(* IEC 61131-3 sources: TIA2AX/tests/V18/test_projects/expected/HW_2000528_main/PLC_LINE_L, 7 files *)

(* ---- HwIdentifiers.st ---- *)
TYPE
	HwIdentifiers : WORD
	(
		PLC_LINE_L_Rail_0 :=	WORD#256,
		PLC_LINE_L :=	WORD#48,
		PLC_LINE_L_Card_reader_writer_1 :=	WORD#51,
		PLC_LINE_L_CPU_display_1 :=	WORD#54,
		PLC_LINE_L_OPC_UA_1 :=	WORD#117,
		PLC_LINE_L_DP_interface_1 :=	WORD#60,
		PLC_LINE_L_PROFINET_interface_1 :=	WORD#64,
		PLC_LINE_L_PROFINET_interface_1_Port_1 :=	WORD#65,
		PLC_LINE_L_PROFINET_interface_1_Port_2 :=	WORD#66,
		PLC_LINE_L_PROFINET_interface_2 :=	WORD#72,
		PLC_LINE_L_PROFINET_interface_2_Port_1 :=	WORD#73,
		UR5_st4_L_Rack :=	WORD#273,
		UR5_st4_L :=	WORD#258,
		UR5_st4_L_Interface :=	WORD#259,
		UR5_st4_L_Interface_RJ45_10_100_MBit_s :=	WORD#260,
		UR5_st4_L_V1_0 :=	WORD#261,
		UR5_st4_L_1_T2O_State :=	WORD#262,
		UR5_st4_L_2_T2O_IO :=	WORD#263,
		UR5_st4_L_3_T2O_Joints :=	WORD#264,
		UR5_st4_L_4_T2O_TCP :=	WORD#265,
		UR5_st4_L_5_T2O_General_Purpose_Bit_Registers :=	WORD#266,
		UR5_st4_L_6_T2O_General_Purpose_Int_Registers :=	WORD#267,
		UR5_st4_L_7_T2O_General_Purpose_Float_Registers :=	WORD#268,
		UR5_st4_L_8_O2T_Robot_IO :=	WORD#269,
		UR5_st4_L_9_O2T_General_Purpose_Registers_1 :=	WORD#270,
		UR5_st4_L_10_O2T_General_Purpose_Registers_2 :=	WORD#271,
		WP001_DM260_L_Rack :=	WORD#275,
		WP001_DM260_L :=	WORD#276,
		WP001_DM260_L_Interface :=	WORD#277,
		WP001_DM260_L_Interface_Port_1 :=	WORD#278,
		WP001_DM260_L_DataMan_260 :=	WORD#279,
		WP001_DM260_L_Acquisition_Control_1 :=	WORD#280,
		WP001_DM260_L_Acquisition_Status_1 :=	WORD#281,
		WP001_DM260_L_Results_Control_1 :=	WORD#282,
		WP001_DM260_L_Results_Status_1 :=	WORD#283,
		WP001_DM260_L_Soft_Event_Control_1 :=	WORD#284,
		WP001_DM260_L_User_Data_64_bytes_1 :=	WORD#285,
		WP001_DM260_L_Result_Data_64_bytes_1 :=	WORD#286,
		R5A1_L_Rack_0 :=	WORD#288,
		R5A1_L :=	WORD#289,
		R5A1_L_R5A1_L :=	WORD#290,
		R5A1_L_PROFINET_interface :=	WORD#291,
		R5A1_L_PROFINET_interface_Port_1 :=	WORD#293,
		R5A1_L_PROFINET_interface_Port_2 :=	WORD#292,
		R5A1_L_BA_2xRJ45 :=	WORD#293,
		R5A1_L_CM_PtP_1 :=	WORD#294,
		R5A1_L_AI_4xU_I_2_wire_ST_1 :=	WORD#295,
		R5A1_L_AI_4xU_I_2_wire_ST_2 :=	WORD#296,
		R5A1_L_AQ_4xU_I_ST_1 :=	WORD#297,
		R5A1_L_DI_16x24VDC_ST_1 :=	WORD#298,
		R5A1_L_DI_16x24VDC_ST_2 :=	WORD#299,
		R5A1_L_DI_16x24VDC_ST_3 :=	WORD#300,
		R5A1_L_DI_16x24VDC_ST_4 :=	WORD#301,
		R5A1_L_DI_16x24VDC_ST_5 :=	WORD#302,
		R5A1_L_DQ_16x24VDC_0_5A_ST_1 :=	WORD#303,
		R5A1_L_DQ_16x24VDC_0_5A_ST_2 :=	WORD#304,
		R5A1_L_DQ_16x24VDC_0_5A_ST_3 :=	WORD#305,
		R5A1_L_DQ_16x24VDC_0_5A_ST_4 :=	WORD#306,
		R5A1_L_TM_Pulse_2x24V_1 :=	WORD#307,
		R5A1_L_TM_Pulse_2x24V_2 :=	WORD#308,
		R5A1_L_Server_module_1 :=	WORD#309,
		R0_L_Rack_0 :=	WORD#311,
		R0_L :=	WORD#312,
		R0_L_R0_L :=	WORD#313,
		R0_L_PROFINET_interface :=	WORD#314,
		R0_L_PROFINET_interface_Port_1 :=	WORD#316,
		R0_L_PROFINET_interface_Port_2 :=	WORD#315,
		R0_L_BA_2xRJ45 :=	WORD#316,
		R0_L_DI_16x24VDC_ST_1 :=	WORD#317,
		R0_L_DI_16x24VDC_ST_2 :=	WORD#318,
		R0_L_DI_16x24VDC_ST_3 :=	WORD#319,
		R0_L_DI_16x24VDC_ST_4 :=	WORD#320,
		R0_L_DI_16x24VDC_ST_5 :=	WORD#321,
		R0_L_DI_16x24VDC_ST_6 :=	WORD#322,
		R0_L_DQ_16x24VDC_0_5A_ST_1 :=	WORD#323,
		R0_L_DQ_16x24VDC_0_5A_ST_2 :=	WORD#324,
		R0_L_DQ_16x24VDC_0_5A_ST_3 :=	WORD#325,
		R0_L_DQ_16x24VDC_0_5A_ST_4 :=	WORD#326,
		R0_L_DQ_16x24VDC_0_5A_ST_5 :=	WORD#327,
		R0_L_DI_8x24VDC_ST_1 :=	WORD#328,
		R0_L_DI_8x24VDC_ST_2 :=	WORD#329,
		R0_L_DI_8x24VDC_ST_3 :=	WORD#330,
		R0_L_DI_8x24VDC_ST_4 :=	WORD#331,
		R0_L_DI_16x24VDC_ST_7 :=	WORD#332,
		R0_L_Server_module_1 :=	WORD#333,
		R1A1_L_Rack_0 :=	WORD#335,
		R1A1_L :=	WORD#336,
		R1A1_L_R1A1_L :=	WORD#337,
		R1A1_L_PROFINET_interface :=	WORD#338,
		R1A1_L_PROFINET_interface_Port_1 :=	WORD#340,
		R1A1_L_PROFINET_interface_Port_2 :=	WORD#339,
		R1A1_L_BA_2xRJ45 :=	WORD#340,
		R1A1_L_DI_16x24VDC_ST_1 :=	WORD#341,
		R1A1_L_DI_16x24VDC_ST_2 :=	WORD#342,
		R1A1_L_DI_16x24VDC_ST_3 :=	WORD#343,
		R1A1_L_DI_16x24VDC_ST_4 :=	WORD#344,
		R1A1_L_DQ_16x24VDC_0_5A_ST_1 :=	WORD#345,
		R1A1_L_DQ_16x24VDC_0_5A_ST_2 :=	WORD#346,
		R1A1_L_DQ_16x24VDC_0_5A_ST_3 :=	WORD#347,
		R1A1_L_Server_module_1 :=	WORD#348,
		R2A1_L_Rack_0 :=	WORD#350,
		R2A1_L :=	WORD#351,
		R2A1_L_R2A1_L :=	WORD#352,
		R2A1_L_PROFINET_interface :=	WORD#353,
		R2A1_L_PROFINET_interface_Port_1 :=	WORD#355,
		R2A1_L_PROFINET_interface_Port_2 :=	WORD#354,
		R2A1_L_BA_2xRJ45 :=	WORD#355,
		R2A1_L_AI_4xU_I_2_wire_ST_1 :=	WORD#356,
		R2A1_L_DI_16x24VDC_ST_1 :=	WORD#357,
		R2A1_L_DI_16x24VDC_ST_2 :=	WORD#358,
		R2A1_L_DI_16x24VDC_ST_3 :=	WORD#359,
		R2A1_L_DI_16x24VDC_ST_4 :=	WORD#360,
		R2A1_L_DI_16x24VDC_ST_5 :=	WORD#361,
		R2A1_L_DI_16x24VDC_ST_6 :=	WORD#362,
		R2A1_L_DQ_16x24VDC_0_5A_ST_1 :=	WORD#363,
		R2A1_L_DQ_16x24VDC_0_5A_ST_2 :=	WORD#364,
		R2A1_L_DQ_16x24VDC_0_5A_ST_3 :=	WORD#365,
		R2A1_L_TM_Pulse_2x24V_1 :=	WORD#366,
		R2A1_L_Server_module_1 :=	WORD#367,
		R6_L_Rack_0 :=	WORD#369,
		R6_L :=	WORD#370,
		R6_L_R6_L :=	WORD#371,
		R6_L_PROFINET_interface :=	WORD#372,
		R6_L_PROFINET_interface_Port_1 :=	WORD#374,
		R6_L_PROFINET_interface_Port_2 :=	WORD#373,
		R6_L_BA_2xRJ45 :=	WORD#374,
		R6_L_DI_16x24VDC_ST_1 :=	WORD#375,
		R6_L_DI_16x24VDC_ST_2 :=	WORD#376,
		R6_L_DQ_16x24VDC_0_5A_ST_1 :=	WORD#377,
		R6_L_DQ_16x24VDC_0_5A_ST_2 :=	WORD#378,
		R6_L_Server_module_1 :=	WORD#379,
		WP002_DM260_L_Rack :=	WORD#381,
		WP002_DM260_L :=	WORD#382,
		WP002_DM260_L_Interface :=	WORD#383,
		WP002_DM260_L_Interface_Port_1 :=	WORD#384,
		WP002_DM260_L_DataMan_260 :=	WORD#385,
		WP002_DM260_L_Acquisition_Control_1 :=	WORD#386,
		WP002_DM260_L_Acquisition_Status_1 :=	WORD#387,
		WP002_DM260_L_Results_Control_1 :=	WORD#388,
		WP002_DM260_L_Results_Status_1 :=	WORD#389,
		WP002_DM260_L_Soft_Event_Control_1 :=	WORD#390,
		WP002_DM260_L_User_Data_64_bytes_1 :=	WORD#391,
		WP002_DM260_L_Result_Data_64_bytes_1 :=	WORD#392,
		CPX_WP5_L_PN_IO_Interface :=	WORD#396,
		CPX_WP5_L_PN_IO_Interface_Port_1 :=	WORD#397,
		CPX_WP5_L_PN_IO_Interface_Port_2 :=	WORD#398,
		CPX_WP5_L_CPX_Rev_30 :=	WORD#399,
		CPX_WP5_L_FB33_PNIO_Module_1 :=	WORD#400,
		CPX_WP5_L_MPA1S_VMPA1_FB_EMS_8_8DO_1 :=	WORD#401,
		CPX_WP5_L_MPA1S_VMPA1_FB_EMS_8_8DO_2 :=	WORD#402,
		CPX_WP5_L_MPA1S_VMPA1_FB_EMS_8_8DO_3 :=	WORD#403,
		CPX_TS_L_PN_IO_Interface :=	WORD#407,
		CPX_TS_L_PN_IO_Interface_Port_1 :=	WORD#408,
		CPX_TS_L_PN_IO_Interface_Port_2 :=	WORD#409,
		CPX_TS_L_CPX_Rev_30 :=	WORD#410,
		CPX_TS_L_FB33_PNIO_Module_1 :=	WORD#411,
		CPX_TS_L_MPA2S_VMPA2_FB_EMS_4_4DO_1 :=	WORD#412,
		CPX_TS_L_MPA2G_VMPA2_FB_EMG_4_4DO_1 :=	WORD#413,
		CPX_TS_L_MPA1G_VMPA1_FB_EMG_8_8DO_2 :=	WORD#414,
		CPX_TS_L_MPA1G_VMPA1_FB_EMG_8_8DO_3 :=	WORD#415,
		CPX_TS_L_MPA1G_VMPA1_FB_EMG_8_8DO_4 :=	WORD#416,
		CPX_TS_L_MPA1G_VMPA1_FB_EMG_8_8DO_5 :=	WORD#417,
		CPX_TS_L_MPA1G_VMPA1_FB_EMG_8_8DO_6 :=	WORD#418,
		CPX_WP2_L_PN_IO_Interface :=	WORD#422,
		CPX_WP2_L_PN_IO_Interface_Port_1 :=	WORD#423,
		CPX_WP2_L_PN_IO_Interface_Port_2 :=	WORD#424,
		CPX_WP2_L_CPX_Rev_30 :=	WORD#425,
		CPX_WP2_L_FB33_PNIO_Module_1 :=	WORD#426,
		CPX_WP2_L_MPA1S_VMPA1_FB_EMS_8_8DO_1 :=	WORD#427,
		CPX_WP2_L_MPA1S_VMPA1_FB_EMS_8_8DO_2 :=	WORD#428,
		CPX_WP2_L_MPA1S_VMPA1_FB_EMS_8_8DO_3 :=	WORD#429,
		CPX_WP2_L_MPA1G_VMPA1_FB_EMG_8_8DO_3 :=	WORD#430,
		fx0_gpnt_L_FX0_GPNT_V2 :=	WORD#434,
		fx0_gpnt_L_FX0_GPNT_V2_Port_1 :=	WORD#435,
		fx0_gpnt_L_FX0_GPNT_V2_Port_2 :=	WORD#436,
		fx0_gpnt_L_FX0_GPNT_V2_1 :=	WORD#437,
		fx0_gpnt_L_Input_Data_Block_1_1 :=	WORD#438,
		fx0_gpnt_L_Input_Data_Block_2_1 :=	WORD#439,
		fx0_gpnt_L_Input_Data_Block_3_1 :=	WORD#440,
		fx0_gpnt_L_Input_Data_Block_4_1 :=	WORD#441,
		fx0_gpnt_L_Input_Data_Block_5_1 :=	WORD#442,
		fx0_gpnt_L_Output_Data_Block_1_1 :=	WORD#443,
		fx0_gpnt_L_Output_Data_Block_2_1 :=	WORD#444,
		fx0_gpnt_L_Output_Data_Block_3_1 :=	WORD#445,
		fx0_gpnt_L_Output_Data_Block_4_1 :=	WORD#446,
		fx0_gpnt_L_Output_Data_Block_5_1 :=	WORD#447,
		WP004_DM260_L_Rack :=	WORD#449,
		WP004_DM260_L :=	WORD#450,
		WP004_DM260_L_Interface :=	WORD#451,
		WP004_DM260_L_Interface_Port_1 :=	WORD#452,
		WP004_DM260_L_DataMan_260 :=	WORD#453,
		WP004_DM260_L_Acquisition_Control_1 :=	WORD#454,
		WP004_DM260_L_Acquisition_Status_1 :=	WORD#455,
		WP004_DM260_L_Results_Control_1 :=	WORD#456,
		WP004_DM260_L_Results_Status_1 :=	WORD#457,
		WP004_DM260_L_Soft_Event_Control_1 :=	WORD#458,
		WP004_DM260_L_User_Data_64_bytes_1 :=	WORD#459,
		WP004_DM260_L_Result_Data_64_bytes_1 :=	WORD#460,
		WP0031_DM260_L_Rack :=	WORD#462,
		WP0031_DM260_L :=	WORD#463,
		WP0031_DM260_L_Interface :=	WORD#464,
		WP0031_DM260_L_Interface_Port_1 :=	WORD#465,
		WP0031_DM260_L_DataMan_260 :=	WORD#466,
		WP0031_DM260_L_Acquisition_Control_1 :=	WORD#467,
		WP0031_DM260_L_Acquisition_Status_1 :=	WORD#468,
		WP0031_DM260_L_Results_Control_1 :=	WORD#469,
		WP0031_DM260_L_Results_Status_1 :=	WORD#470,
		WP0031_DM260_L_Soft_Event_Control_1 :=	WORD#471,
		WP0031_DM260_L_User_Data_64_bytes_1 :=	WORD#472,
		WP0031_DM260_L_Result_Data_64_bytes_1 :=	WORD#473,
		WP003_DM260_L_Rack :=	WORD#475,
		WP003_DM260_L :=	WORD#476,
		WP003_DM260_L_Interface :=	WORD#477,
		WP003_DM260_L_Interface_Port_1 :=	WORD#478,
		WP003_DM260_L_DataMan_260 :=	WORD#479,
		WP003_DM260_L_Acquisition_Control_1 :=	WORD#480,
		WP003_DM260_L_Acquisition_Status_1 :=	WORD#481,
		WP003_DM260_L_Results_Control_1 :=	WORD#482,
		WP003_DM260_L_Results_Status_1 :=	WORD#483,
		WP003_DM260_L_Soft_Event_Control_1 :=	WORD#484,
		WP003_DM260_L_User_Data_64_bytes_1 :=	WORD#485,
		WP003_DM260_L_Result_Data_64_bytes_1 :=	WORD#486,
		WP005_DM260_L_Rack :=	WORD#488,
		WP005_DM260_L :=	WORD#489,
		WP005_DM260_L_Interface :=	WORD#490,
		WP005_DM260_L_Interface_Port_1 :=	WORD#491,
		WP005_DM260_L_DataMan_260 :=	WORD#492,
		WP005_DM260_L_Acquisition_Control_1 :=	WORD#493,
		WP005_DM260_L_Acquisition_Status_1 :=	WORD#494,
		WP005_DM260_L_Results_Control_1 :=	WORD#495,
		WP005_DM260_L_Results_Status_1 :=	WORD#496,
		WP005_DM260_L_Soft_Event_Control_1 :=	WORD#497,
		WP005_DM260_L_User_Data_64_bytes_1 :=	WORD#498,
		WP005_DM260_L_Result_Data_64_bytes_1 :=	WORD#499,
		WP006_DM260_L_Rack :=	WORD#501,
		WP006_DM260_L :=	WORD#502,
		WP006_DM260_L_Interface :=	WORD#503,
		WP006_DM260_L_Interface_Port_1 :=	WORD#504,
		WP006_DM260_L_DataMan_260 :=	WORD#505,
		WP006_DM260_L_Acquisition_Control_1 :=	WORD#506,
		WP006_DM260_L_Acquisition_Status_1 :=	WORD#507,
		WP006_DM260_L_Results_Control_1 :=	WORD#508,
		WP006_DM260_L_Results_Status_1 :=	WORD#509,
		WP006_DM260_L_Soft_Event_Control_1 :=	WORD#510,
		WP006_DM260_L_User_Data_64_bytes_1 :=	WORD#511,
		WP006_DM260_L_Result_Data_64_bytes_1 :=	WORD#512,
		WP001_DM8050_L_Rack :=	WORD#514,
		WP001_DM8050_L :=	WORD#515,
		WP001_DM8050_L_Interface :=	WORD#516,
		WP001_DM8050_L_Interface_Port_1 :=	WORD#517,
		WP001_DM8050_L_DataMan_8000 :=	WORD#518,
		WP001_DM8050_L_Acquisition_Control_1 :=	WORD#519,
		WP001_DM8050_L_Acquisition_Status_1 :=	WORD#520,
		WP001_DM8050_L_Results_Control_1 :=	WORD#521,
		WP001_DM8050_L_Results_Status_1 :=	WORD#522,
		WP001_DM8050_L_Soft_Event_Control_1 :=	WORD#523,
		WP001_DM8050_L_User_Data_64_bytes_1 :=	WORD#524,
		WP001_DM8050_L_Result_Data_64_bytes_1 :=	WORD#525,
		WP004_DM8050_L_Rack :=	WORD#527,
		WP004_DM8050_L :=	WORD#528,
		WP004_DM8050_L_Interface :=	WORD#529,
		WP004_DM8050_L_Interface_Port_1 :=	WORD#530,
		WP004_DM8050_L_DataMan_8000 :=	WORD#531,
		WP004_DM8050_L_Acquisition_Control_1 :=	WORD#532,
		WP004_DM8050_L_Acquisition_Status_1 :=	WORD#533,
		WP004_DM8050_L_Results_Control_1 :=	WORD#534,
		WP004_DM8050_L_Results_Status_1 :=	WORD#535,
		WP004_DM8050_L_Soft_Event_Control_1 :=	WORD#536,
		WP004_DM8050_L_User_Data_64_bytes_1 :=	WORD#537,
		WP004_DM8050_L_Result_Data_64_bytes_1 :=	WORD#538,
		WP003_CAM_L_Rack :=	WORD#540,
		WP003_CAM_L :=	WORD#541,
		WP003_CAM_L_Interface :=	WORD#542,
		WP003_CAM_L_Interface_Port_1 :=	WORD#543,
		WP003_CAM_L_In_Sight_IS2XXX_CC_B :=	WORD#544,
		WP003_CAM_L_Acquisition_Control_1 :=	WORD#545,
		WP003_CAM_L_Acquisition_Status_1 :=	WORD#546,
		WP003_CAM_L_Inspection_Control_1 :=	WORD#547,
		WP003_CAM_L_Inspection_Status_1 :=	WORD#548,
		WP003_CAM_L_Command_Control_1 :=	WORD#549,
		WP003_CAM_L_SoftEvent_Control_1 :=	WORD#550,
		WP003_CAM_L_User_Data_64_bytes_1 :=	WORD#551,
		WP003_CAM_L_Results_64_bytes_1 :=	WORD#552,
		WP004_CAM_L_Rack :=	WORD#554,
		WP004_CAM_L :=	WORD#555,
		WP004_CAM_L_Interface :=	WORD#556,
		WP004_CAM_L_Interface_Port_1 :=	WORD#557,
		WP004_CAM_L_In_Sight_IS2XXX_CC_B :=	WORD#558,
		WP004_CAM_L_Acquisition_Control_1 :=	WORD#559,
		WP004_CAM_L_Acquisition_Status_1 :=	WORD#560,
		WP004_CAM_L_Inspection_Control_1 :=	WORD#561,
		WP004_CAM_L_Inspection_Status_1 :=	WORD#562,
		WP004_CAM_L_Command_Control_1 :=	WORD#563,
		WP004_CAM_L_SoftEvent_Control_1 :=	WORD#564,
		WP004_CAM_L_User_Data_64_bytes_1 :=	WORD#565,
		WP004_CAM_L_Results_64_bytes_1 :=	WORD#566,
		WP0031_DM8700_L_Rack :=	WORD#568,
		WP0031_DM8700_L :=	WORD#569,
		WP0031_DM8700_L_Interface :=	WORD#570,
		WP0031_DM8700_L_Interface_Port_1 :=	WORD#571,
		WP0031_DM8700_L_DataMan_8700_CC_B :=	WORD#572,
		WP0031_DM8700_L_Acquisition_Control_1 :=	WORD#573,
		WP0031_DM8700_L_Acquisition_Status_1 :=	WORD#574,
		WP0031_DM8700_L_Results_Control_1 :=	WORD#575,
		WP0031_DM8700_L_Results_Status_1 :=	WORD#576,
		WP0031_DM8700_L_Soft_Event_Control_1 :=	WORD#577,
		WP0031_DM8700_L_User_Data_64_bytes_1 :=	WORD#578,
		WP0031_DM8700_L_Result_Data_64_bytes_1 :=	WORD#579,
		WP002_DM8050_L_Rack :=	WORD#581,
		WP002_DM8050_L :=	WORD#582,
		WP002_DM8050_L_Interface :=	WORD#583,
		WP002_DM8050_L_Interface_Port_1 :=	WORD#584,
		WP002_DM8050_L_DataMan_8000 :=	WORD#585,
		WP002_DM8050_L_Acquisition_Control_1 :=	WORD#586,
		WP002_DM8050_L_Acquisition_Status_1 :=	WORD#587,
		WP002_DM8050_L_Results_Control_1 :=	WORD#588,
		WP002_DM8050_L_Results_Status_1 :=	WORD#589,
		WP002_DM8050_L_Soft_Event_Control_1 :=	WORD#590,
		WP002_DM8050_L_User_Data_64_bytes_1 :=	WORD#591,
		WP002_DM8050_L_Result_Data_64_bytes_1 :=	WORD#592,
		CPX_Rack_L_PN_IO_Interface :=	WORD#596,
		CPX_Rack_L_PN_IO_Interface_Port_1 :=	WORD#597,
		CPX_Rack_L_PN_IO_Interface_Port_2 :=	WORD#598,
		CPX_Rack_L_CPX_Rev_30 :=	WORD#599,
		CPX_Rack_L_FB33_PNIO_Module_1 :=	WORD#600,
		CPX_Rack_L_16DI_16DI_1 :=	WORD#601,
		CPX_Rack_L_16DI_16DI_2 :=	WORD#602,
		CPX_Rack_L_16DI_16DI_3 :=	WORD#603,
		CPX_Rack_L_16DI_16DI_4 :=	WORD#604,
		CPX_Rack_L_16DI_16DI_5 :=	WORD#605,
		CPX_Rack_L_MPA1S_VMPA1_FB_EMS_8_8DO_1 :=	WORD#606,
		CPX_Rack_L_MPA1S_VMPA1_FB_EMS_8_8DO_2 :=	WORD#607,
		CPX_Rack_L_MPA1S_VMPA1_FB_EMS_8_8DO_3 :=	WORD#608,
		CPX_Rack_L_MPA1S_VMPA1_FB_EMS_8_8DO_4 :=	WORD#609,
		CPX_Rack_L_MPA1S_VMPA1_FB_EMS_8_8DO_5 :=	WORD#610,
		WP000_DM260_L_Rack :=	WORD#612,
		WP000_DM260_L :=	WORD#613,
		WP000_DM260_L_Interface :=	WORD#614,
		WP000_DM260_L_Interface_Port_1 :=	WORD#615,
		WP000_DM260_L_DataMan_260 :=	WORD#616,
		WP000_DM260_L_Acquisition_Control_1 :=	WORD#617,
		WP000_DM260_L_Acquisition_Status_1 :=	WORD#618,
		WP000_DM260_L_Results_Control_1 :=	WORD#619,
		WP000_DM260_L_Results_Status_1 :=	WORD#620,
		WP000_DM260_L_Soft_Event_Control_1 :=	WORD#621,
		WP000_DM260_L_User_Data_64_bytes_1 :=	WORD#622,
		WP000_DM260_L_Result_Data_64_bytes_1 :=	WORD#623,
		WP000_DM8050_L_Rack :=	WORD#625,
		WP000_DM8050_L :=	WORD#626,
		WP000_DM8050_L_Interface :=	WORD#627,
		WP000_DM8050_L_Interface_Port_1 :=	WORD#628,
		WP000_DM8050_L_DataMan_8000 :=	WORD#629,
		WP000_DM8050_L_Acquisition_Control_1 :=	WORD#630,
		WP000_DM8050_L_Acquisition_Status_1 :=	WORD#631,
		WP000_DM8050_L_Results_Control_1 :=	WORD#632,
		WP000_DM8050_L_Results_Status_1 :=	WORD#633,
		WP000_DM8050_L_Soft_Event_Control_1 :=	WORD#634,
		WP000_DM8050_L_User_Data_64_bytes_1 :=	WORD#635,
		WP000_DM8050_L_Result_Data_64_bytes_1 :=	WORD#636,
		NONE:= WORD#0
	);
END_TYPE

(* ---- HwInputs.st ---- *)
TYPE
	HwInputs : STRUCT
		UR5_st4_L_1_T2O_State AT %B1080 : ARRAY[0..31] OF BYTE;
		UR5_st4_L_2_T2O_IO AT %B1112 : ARRAY[0..67] OF BYTE;
		UR5_st4_L_3_T2O_Joints AT %B2696 : ARRAY[0..103] OF BYTE;
		UR5_st4_L_4_T2O_TCP AT %B1304 : ARRAY[0..75] OF BYTE;
		UR5_st4_L_5_T2O_General_Purpose_Bit_Registers AT %B1380 : ARRAY[0..7] OF BYTE;
		UR5_st4_L_6_T2O_General_Purpose_Int_Registers AT %B2800 : ARRAY[0..95] OF BYTE;
		UR5_st4_L_7_T2O_General_Purpose_Float_Registers AT %B2896 : ARRAY[0..95] OF BYTE;
		WP001_DM260_L_Acquisition_Status_1 AT %B5100 : ARRAY[0..2] OF BYTE;
		WP001_DM260_L_Results_Status_1 AT %B5103 : BYTE;
		WP001_DM260_L_Soft_Event_Control_1 AT %B5104 : BYTE;
		WP001_DM260_L_Result_Data_64_bytes_1 AT %B5110 : ARRAY[0..71] OF BYTE;
		R5A1_L_CM_PtP_1 AT %B270 : ARRAY[0..7] OF BYTE;
		R5A1_L_AI_4xU_I_2_wire_ST_1 AT %B278 : ARRAY[0..7] OF BYTE;
		R5A1_L_AI_4xU_I_2_wire_ST_2 AT %B286 : ARRAY[0..7] OF BYTE;
		R5A1_L_DI_16x24VDC_ST_1 AT %B20 : WORD;
		R5A1_L_DI_16x24VDC_ST_2 AT %B22 : WORD;
		R5A1_L_DI_16x24VDC_ST_3 AT %B24 : WORD;
		R5A1_L_DI_16x24VDC_ST_4 AT %B26 : WORD;
		R5A1_L_DI_16x24VDC_ST_5 AT %B28 : WORD;
		R5A1_L_TM_Pulse_2x24V_1 AT %B224 : ARRAY[0..15] OF BYTE;
		R5A1_L_TM_Pulse_2x24V_2 AT %B250 : ARRAY[0..15] OF BYTE;
		R0_L_DI_16x24VDC_ST_1 AT %B0 : WORD;
		R0_L_DI_16x24VDC_ST_2 AT %B2 : WORD;
		R0_L_DI_16x24VDC_ST_3 AT %B4 : WORD;
		R0_L_DI_16x24VDC_ST_4 AT %B6 : WORD;
		R0_L_DI_16x24VDC_ST_5 AT %B8 : WORD;
		R0_L_DI_16x24VDC_ST_6 AT %B10 : WORD;
		R0_L_DI_8x24VDC_ST_1 AT %B12 : BYTE;
		R0_L_DI_8x24VDC_ST_2 AT %B13 : BYTE;
		R0_L_DI_8x24VDC_ST_3 AT %B14 : BYTE;
		R0_L_DI_8x24VDC_ST_4 AT %B15 : BYTE;
		R0_L_DI_16x24VDC_ST_7 AT %B16 : WORD;
		R1A1_L_DI_16x24VDC_ST_1 AT %B100 : WORD;
		R1A1_L_DI_16x24VDC_ST_2 AT %B102 : WORD;
		R1A1_L_DI_16x24VDC_ST_3 AT %B104 : WORD;
		R1A1_L_DI_16x24VDC_ST_4 AT %B106 : WORD;
		R2A1_L_AI_4xU_I_2_wire_ST_1 AT %B2000 : ARRAY[0..7] OF BYTE;
		R2A1_L_DI_16x24VDC_ST_1 AT %B200 : WORD;
		R2A1_L_DI_16x24VDC_ST_2 AT %B202 : WORD;
		R2A1_L_DI_16x24VDC_ST_3 AT %B204 : WORD;
		R2A1_L_DI_16x24VDC_ST_4 AT %B206 : WORD;
		R2A1_L_DI_16x24VDC_ST_5 AT %B208 : WORD;
		R2A1_L_DI_16x24VDC_ST_6 AT %B210 : WORD;
		R2A1_L_TM_Pulse_2x24V_1 AT %B2010 : ARRAY[0..15] OF BYTE;
		R6_L_DI_16x24VDC_ST_1 AT %B600 : WORD;
		R6_L_DI_16x24VDC_ST_2 AT %B602 : WORD;
		WP002_DM260_L_Acquisition_Status_1 AT %B5105 : ARRAY[0..2] OF BYTE;
		WP002_DM260_L_Results_Status_1 AT %B5108 : BYTE;
		WP002_DM260_L_Soft_Event_Control_1 AT %B5109 : BYTE;
		WP002_DM260_L_Result_Data_64_bytes_1 AT %B5182 : ARRAY[0..71] OF BYTE;
		fx0_gpnt_L_Input_Data_Block_1_1 AT %B950 : ARRAY[0..11] OF BYTE;
		fx0_gpnt_L_Input_Data_Block_2_1 AT %B962 : ARRAY[0..11] OF BYTE;
		fx0_gpnt_L_Input_Data_Block_3_1 AT %B974 : ARRAY[0..11] OF BYTE;
		fx0_gpnt_L_Input_Data_Block_4_1 AT %B986 : ARRAY[0..11] OF BYTE;
		fx0_gpnt_L_Input_Data_Block_5_1 AT %B998 : WORD;
		WP004_DM260_L_Acquisition_Status_1 AT %B5408 : ARRAY[0..2] OF BYTE;
		WP004_DM260_L_Results_Status_1 AT %B5411 : BYTE;
		WP004_DM260_L_Soft_Event_Control_1 AT %B5412 : BYTE;
		WP004_DM260_L_Result_Data_64_bytes_1 AT %B5413 : ARRAY[0..71] OF BYTE;
		WP0031_DM260_L_Acquisition_Status_1 AT %B5485 : ARRAY[0..2] OF BYTE;
		WP0031_DM260_L_Results_Status_1 AT %B5488 : BYTE;
		WP0031_DM260_L_Soft_Event_Control_1 AT %B5489 : BYTE;
		WP0031_DM260_L_Result_Data_64_bytes_1 AT %B5490 : ARRAY[0..71] OF BYTE;
		WP003_DM260_L_Acquisition_Status_1 AT %B5562 : ARRAY[0..2] OF BYTE;
		WP003_DM260_L_Results_Status_1 AT %B5565 : BYTE;
		WP003_DM260_L_Soft_Event_Control_1 AT %B5566 : BYTE;
		WP003_DM260_L_Result_Data_64_bytes_1 AT %B5567 : ARRAY[0..71] OF BYTE;
		WP005_DM260_L_Acquisition_Status_1 AT %B5331 : ARRAY[0..2] OF BYTE;
		WP005_DM260_L_Results_Status_1 AT %B5334 : BYTE;
		WP005_DM260_L_Soft_Event_Control_1 AT %B5335 : BYTE;
		WP005_DM260_L_Result_Data_64_bytes_1 AT %B5336 : ARRAY[0..71] OF BYTE;
		WP006_DM260_L_Acquisition_Status_1 AT %B5254 : ARRAY[0..2] OF BYTE;
		WP006_DM260_L_Results_Status_1 AT %B5257 : BYTE;
		WP006_DM260_L_Soft_Event_Control_1 AT %B5258 : BYTE;
		WP006_DM260_L_Result_Data_64_bytes_1 AT %B5259 : ARRAY[0..71] OF BYTE;
		WP001_DM8050_L_Acquisition_Status_1 AT %B46 : ARRAY[0..2] OF BYTE;
		WP001_DM8050_L_Results_Status_1 AT %B49 : BYTE;
		WP001_DM8050_L_Soft_Event_Control_1 AT %B50 : BYTE;
		WP001_DM8050_L_Result_Data_64_bytes_1 AT %B362 : ARRAY[0..71] OF BYTE;
		WP004_DM8050_L_Acquisition_Status_1 AT %B56 : ARRAY[0..2] OF BYTE;
		WP004_DM8050_L_Results_Status_1 AT %B59 : BYTE;
		WP004_DM8050_L_Soft_Event_Control_1 AT %B60 : BYTE;
		WP004_DM8050_L_Result_Data_64_bytes_1 AT %B506 : ARRAY[0..71] OF BYTE;
		WP003_CAM_L_Acquisition_Status_1 AT %B30 : ARRAY[0..2] OF BYTE;
		WP003_CAM_L_Inspection_Status_1 AT %B61 : DWORD;
		WP003_CAM_L_Command_Control_1 AT %B18 : WORD;
		WP003_CAM_L_SoftEvent_Control_1 AT %B33 : BYTE;
		WP003_CAM_L_Results_64_bytes_1 AT %B108 : ARRAY[0..67] OF BYTE;
		WP004_CAM_L_Acquisition_Status_1 AT %B34 : ARRAY[0..2] OF BYTE;
		WP004_CAM_L_Inspection_Status_1 AT %B37 : DWORD;
		WP004_CAM_L_Command_Control_1 AT %B41 : WORD;
		WP004_CAM_L_SoftEvent_Control_1 AT %B43 : BYTE;
		WP004_CAM_L_Results_64_bytes_1 AT %B294 : ARRAY[0..67] OF BYTE;
		WP0031_DM8700_L_Acquisition_Status_1 AT %B51 : ARRAY[0..2] OF BYTE;
		WP0031_DM8700_L_Results_Status_1 AT %B44 : BYTE;
		WP0031_DM8700_L_Soft_Event_Control_1 AT %B45 : BYTE;
		WP0031_DM8700_L_Result_Data_64_bytes_1 AT %B434 : ARRAY[0..71] OF BYTE;
		WP002_DM8050_L_Acquisition_Status_1 AT %B65 : ARRAY[0..2] OF BYTE;
		WP002_DM8050_L_Results_Status_1 AT %B54 : BYTE;
		WP002_DM8050_L_Soft_Event_Control_1 AT %B55 : BYTE;
		WP002_DM8050_L_Result_Data_64_bytes_1 AT %B604 : ARRAY[0..71] OF BYTE;
		CPX_Rack_L_16DI_16DI_1 AT %B80 : WORD;
		CPX_Rack_L_16DI_16DI_2 AT %B82 : WORD;
		CPX_Rack_L_16DI_16DI_3 AT %B84 : WORD;
		CPX_Rack_L_16DI_16DI_4 AT %B86 : WORD;
		CPX_Rack_L_16DI_16DI_5 AT %B88 : WORD;
		WP000_DM260_L_Acquisition_Status_1 AT %B5639 : ARRAY[0..2] OF BYTE;
		WP000_DM260_L_Results_Status_1 AT %B5642 : BYTE;
		WP000_DM260_L_Soft_Event_Control_1 AT %B5643 : BYTE;
		WP000_DM260_L_Result_Data_64_bytes_1 AT %B5644 : ARRAY[0..71] OF BYTE;
		WP000_DM8050_L_Acquisition_Status_1 AT %B68 : ARRAY[0..2] OF BYTE;
		WP000_DM8050_L_Results_Status_1 AT %B71 : BYTE;
		WP000_DM8050_L_Soft_Event_Control_1 AT %B72 : BYTE;
		WP000_DM8050_L_Result_Data_64_bytes_1 AT %B676 : ARRAY[0..71] OF BYTE;
	END_STRUCT;
END_TYPE

(* ---- HwOutputs.st ---- *)
TYPE
	HwOutputs : STRUCT
		UR5_st4_L_8_O2T_Robot_IO AT %B874 : ARRAY[0..23] OF BYTE;
		UR5_st4_L_9_O2T_General_Purpose_Registers_1 AT %B1070 : ARRAY[0..99] OF BYTE;
		UR5_st4_L_10_O2T_General_Purpose_Registers_2 AT %B2502 : ARRAY[0..99] OF BYTE;
		WP001_DM260_L_Acquisition_Control_1 AT %B5100 : BYTE;
		WP001_DM260_L_Results_Control_1 AT %B5101 : BYTE;
		WP001_DM260_L_Soft_Event_Control_1 AT %B5104 : BYTE;
		WP001_DM260_L_User_Data_64_bytes_1 AT %B5110 : ARRAY[0..67] OF BYTE;
		R5A1_L_AQ_4xU_I_ST_1 AT %B280 : ARRAY[0..7] OF BYTE;
		R5A1_L_DQ_16x24VDC_0_5A_ST_1 AT %B20 : WORD;
		R5A1_L_DQ_16x24VDC_0_5A_ST_2 AT %B22 : WORD;
		R5A1_L_DQ_16x24VDC_0_5A_ST_3 AT %B24 : WORD;
		R5A1_L_DQ_16x24VDC_0_5A_ST_4 AT %B26 : WORD;
		R5A1_L_TM_Pulse_2x24V_1 AT %B224 : ARRAY[0..23] OF BYTE;
		R5A1_L_TM_Pulse_2x24V_2 AT %B250 : ARRAY[0..23] OF BYTE;
		R0_L_DQ_16x24VDC_0_5A_ST_1 AT %B0 : WORD;
		R0_L_DQ_16x24VDC_0_5A_ST_2 AT %B2 : WORD;
		R0_L_DQ_16x24VDC_0_5A_ST_3 AT %B4 : WORD;
		R0_L_DQ_16x24VDC_0_5A_ST_4 AT %B6 : WORD;
		R0_L_DQ_16x24VDC_0_5A_ST_5 AT %B8 : WORD;
		R1A1_L_DQ_16x24VDC_0_5A_ST_1 AT %B100 : WORD;
		R1A1_L_DQ_16x24VDC_0_5A_ST_2 AT %B102 : WORD;
		R1A1_L_DQ_16x24VDC_0_5A_ST_3 AT %B104 : WORD;
		R2A1_L_DQ_16x24VDC_0_5A_ST_1 AT %B200 : WORD;
		R2A1_L_DQ_16x24VDC_0_5A_ST_2 AT %B202 : WORD;
		R2A1_L_DQ_16x24VDC_0_5A_ST_3 AT %B204 : WORD;
		R2A1_L_TM_Pulse_2x24V_1 AT %B2010 : ARRAY[0..23] OF BYTE;
		R6_L_DQ_16x24VDC_0_5A_ST_1 AT %B600 : WORD;
		R6_L_DQ_16x24VDC_0_5A_ST_2 AT %B602 : WORD;
		WP002_DM260_L_Acquisition_Control_1 AT %B5102 : BYTE;
		WP002_DM260_L_Results_Control_1 AT %B5103 : BYTE;
		WP002_DM260_L_Soft_Event_Control_1 AT %B5105 : BYTE;
		WP002_DM260_L_User_Data_64_bytes_1 AT %B5178 : ARRAY[0..67] OF BYTE;
		CPX_WP5_L_MPA1S_VMPA1_FB_EMS_8_8DO_1 AT %B80 : BYTE;
		CPX_WP5_L_MPA1S_VMPA1_FB_EMS_8_8DO_2 AT %B81 : BYTE;
		CPX_WP5_L_MPA1S_VMPA1_FB_EMS_8_8DO_3 AT %B82 : BYTE;
		CPX_TS_L_MPA2S_VMPA2_FB_EMS_4_4DO_1 AT %B50 : BYTE;
		CPX_TS_L_MPA2G_VMPA2_FB_EMG_4_4DO_1 AT %B51 : BYTE;
		CPX_TS_L_MPA1G_VMPA1_FB_EMG_8_8DO_2 AT %B52 : BYTE;
		CPX_TS_L_MPA1G_VMPA1_FB_EMG_8_8DO_3 AT %B53 : BYTE;
		CPX_TS_L_MPA1G_VMPA1_FB_EMG_8_8DO_4 AT %B54 : BYTE;
		CPX_TS_L_MPA1G_VMPA1_FB_EMG_8_8DO_5 AT %B55 : BYTE;
		CPX_TS_L_MPA1G_VMPA1_FB_EMG_8_8DO_6 AT %B56 : BYTE;
		CPX_WP2_L_MPA1S_VMPA1_FB_EMS_8_8DO_1 AT %B60 : BYTE;
		CPX_WP2_L_MPA1S_VMPA1_FB_EMS_8_8DO_2 AT %B61 : BYTE;
		CPX_WP2_L_MPA1S_VMPA1_FB_EMS_8_8DO_3 AT %B62 : BYTE;
		CPX_WP2_L_MPA1G_VMPA1_FB_EMG_8_8DO_3 AT %B63 : BYTE;
		fx0_gpnt_L_Output_Data_Block_1_1 AT %B950 : ARRAY[0..9] OF BYTE;
		fx0_gpnt_L_Output_Data_Block_2_1 AT %B960 : ARRAY[0..9] OF BYTE;
		fx0_gpnt_L_Output_Data_Block_3_1 AT %B970 : ARRAY[0..9] OF BYTE;
		fx0_gpnt_L_Output_Data_Block_4_1 AT %B980 : ARRAY[0..9] OF BYTE;
		fx0_gpnt_L_Output_Data_Block_5_1 AT %B990 : ARRAY[0..9] OF BYTE;
		WP004_DM260_L_Acquisition_Control_1 AT %B5384 : BYTE;
		WP004_DM260_L_Results_Control_1 AT %B5385 : BYTE;
		WP004_DM260_L_Soft_Event_Control_1 AT %B5386 : BYTE;
		WP004_DM260_L_User_Data_64_bytes_1 AT %B5387 : ARRAY[0..67] OF BYTE;
		WP0031_DM260_L_Acquisition_Control_1 AT %B5455 : BYTE;
		WP0031_DM260_L_Results_Control_1 AT %B5456 : BYTE;
		WP0031_DM260_L_Soft_Event_Control_1 AT %B5457 : BYTE;
		WP0031_DM260_L_User_Data_64_bytes_1 AT %B5458 : ARRAY[0..67] OF BYTE;
		WP003_DM260_L_Acquisition_Control_1 AT %B5526 : BYTE;
		WP003_DM260_L_Results_Control_1 AT %B5527 : BYTE;
		WP003_DM260_L_Soft_Event_Control_1 AT %B5528 : BYTE;
		WP003_DM260_L_User_Data_64_bytes_1 AT %B5529 : ARRAY[0..67] OF BYTE;
		WP005_DM260_L_Acquisition_Control_1 AT %B5109 : BYTE;
		WP005_DM260_L_Results_Control_1 AT %B5314 : BYTE;
		WP005_DM260_L_Soft_Event_Control_1 AT %B5315 : BYTE;
		WP005_DM260_L_User_Data_64_bytes_1 AT %B5316 : ARRAY[0..67] OF BYTE;
		WP006_DM260_L_Acquisition_Control_1 AT %B5106 : BYTE;
		WP006_DM260_L_Results_Control_1 AT %B5107 : BYTE;
		WP006_DM260_L_Soft_Event_Control_1 AT %B5108 : BYTE;
		WP006_DM260_L_User_Data_64_bytes_1 AT %B5246 : ARRAY[0..67] OF BYTE;
		WP001_DM8050_L_Acquisition_Control_1 AT %B28 : BYTE;
		WP001_DM8050_L_Results_Control_1 AT %B29 : BYTE;
		WP001_DM8050_L_Soft_Event_Control_1 AT %B30 : BYTE;
		WP001_DM8050_L_User_Data_64_bytes_1 AT %B352 : ARRAY[0..67] OF BYTE;
		WP004_DM8050_L_Acquisition_Control_1 AT %B34 : BYTE;
		WP004_DM8050_L_Results_Control_1 AT %B35 : BYTE;
		WP004_DM8050_L_Soft_Event_Control_1 AT %B36 : BYTE;
		WP004_DM8050_L_User_Data_64_bytes_1 AT %B488 : ARRAY[0..67] OF BYTE;
		WP003_CAM_L_Acquisition_Control_1 AT %B10 : BYTE;
		WP003_CAM_L_Inspection_Control_1 AT %B11 : BYTE;
		WP003_CAM_L_Command_Control_1 AT %B12 : WORD;
		WP003_CAM_L_SoftEvent_Control_1 AT %B14 : BYTE;
		WP003_CAM_L_User_Data_64_bytes_1 AT %B106 : ARRAY[0..63] OF BYTE;
		WP004_CAM_L_Acquisition_Control_1 AT %B15 : BYTE;
		WP004_CAM_L_Inspection_Control_1 AT %B16 : BYTE;
		WP004_CAM_L_Command_Control_1 AT %B17 : WORD;
		WP004_CAM_L_SoftEvent_Control_1 AT %B19 : BYTE;
		WP004_CAM_L_User_Data_64_bytes_1 AT %B288 : ARRAY[0..63] OF BYTE;
		WP0031_DM8700_L_Acquisition_Control_1 AT %B31 : BYTE;
		WP0031_DM8700_L_Results_Control_1 AT %B32 : BYTE;
		WP0031_DM8700_L_Soft_Event_Control_1 AT %B33 : BYTE;
		WP0031_DM8700_L_User_Data_64_bytes_1 AT %B420 : ARRAY[0..67] OF BYTE;
		WP002_DM8050_L_Acquisition_Control_1 AT %B37 : BYTE;
		WP002_DM8050_L_Results_Control_1 AT %B38 : BYTE;
		WP002_DM8050_L_Soft_Event_Control_1 AT %B39 : BYTE;
		WP002_DM8050_L_User_Data_64_bytes_1 AT %B604 : ARRAY[0..67] OF BYTE;
		CPX_Rack_L_MPA1S_VMPA1_FB_EMS_8_8DO_1 AT %B40 : BYTE;
		CPX_Rack_L_MPA1S_VMPA1_FB_EMS_8_8DO_2 AT %B41 : BYTE;
		CPX_Rack_L_MPA1S_VMPA1_FB_EMS_8_8DO_3 AT %B42 : BYTE;
		CPX_Rack_L_MPA1S_VMPA1_FB_EMS_8_8DO_4 AT %B43 : BYTE;
		CPX_Rack_L_MPA1S_VMPA1_FB_EMS_8_8DO_5 AT %B44 : BYTE;
		WP000_DM260_L_Acquisition_Control_1 AT %B5597 : BYTE;
		WP000_DM260_L_Results_Control_1 AT %B5598 : BYTE;
		WP000_DM260_L_Soft_Event_Control_1 AT %B5599 : BYTE;
		WP000_DM260_L_User_Data_64_bytes_1 AT %B5600 : ARRAY[0..67] OF BYTE;
		WP000_DM8050_L_Acquisition_Control_1 AT %B45 : BYTE;
		WP000_DM8050_L_Results_Control_1 AT %B46 : BYTE;
		WP000_DM8050_L_Soft_Event_Control_1 AT %B47 : BYTE;
		WP000_DM8050_L_User_Data_64_bytes_1 AT %B672 : ARRAY[0..67] OF BYTE;
	END_STRUCT;
END_TYPE

(* ---- PlcInputs.st ---- *)
TYPE
	PlcInputs : STRUCT
		UR5_st4_L_1_T2O_State : ARRAY[0..31] OF BYTE;
		UR5_st4_L_2_T2O_IO : ARRAY[0..67] OF BYTE;
		UR5_st4_L_3_T2O_Joints : ARRAY[0..103] OF BYTE;
		UR5_st4_L_4_T2O_TCP : ARRAY[0..75] OF BYTE;
		UR5_st4_L_5_T2O_General_Purpose_Bit_Registers : ARRAY[0..7] OF BYTE;
		UR5_st4_L_6_T2O_General_Purpose_Int_Registers : ARRAY[0..95] OF BYTE;
		UR5_st4_L_7_T2O_General_Purpose_Float_Registers : ARRAY[0..95] OF BYTE;
		WP001_DM260_L_Acquisition_Status_1 : ARRAY[0..2] OF BYTE;
		WP001_DM260_L_Results_Status_1 : BYTE;
		WP001_DM260_L_Soft_Event_Control_1 : BYTE;
		WP001_DM260_L_Result_Data_64_bytes_1 : ARRAY[0..71] OF BYTE;
		R5A1_L_CM_PtP_1 : ARRAY[0..7] OF BYTE;
		R5A1_L_AI_4xU_I_2_wire_ST_1 : ARRAY[0..7] OF BYTE;
		R5A1_L_AI_4xU_I_2_wire_ST_2 : ARRAY[0..7] OF BYTE;
		R5A1_L_DI_16x24VDC_ST_1 : WORD;
		R5A1_L_DI_16x24VDC_ST_2 : WORD;
		R5A1_L_DI_16x24VDC_ST_3 : WORD;
		R5A1_L_DI_16x24VDC_ST_4 : WORD;
		R5A1_L_DI_16x24VDC_ST_5 : WORD;
		R5A1_L_TM_Pulse_2x24V_1 : ARRAY[0..15] OF BYTE;
		R5A1_L_TM_Pulse_2x24V_2 : ARRAY[0..15] OF BYTE;
		R0_L_DI_16x24VDC_ST_1 : WORD;
		R0_L_DI_16x24VDC_ST_2 : WORD;
		R0_L_DI_16x24VDC_ST_3 : WORD;
		R0_L_DI_16x24VDC_ST_4 : WORD;
		R0_L_DI_16x24VDC_ST_5 : WORD;
		R0_L_DI_16x24VDC_ST_6 : WORD;
		R0_L_DI_8x24VDC_ST_1 : BYTE;
		R0_L_DI_8x24VDC_ST_2 : BYTE;
		R0_L_DI_8x24VDC_ST_3 : BYTE;
		R0_L_DI_8x24VDC_ST_4 : BYTE;
		R0_L_DI_16x24VDC_ST_7 : WORD;
		R1A1_L_DI_16x24VDC_ST_1 : WORD;
		R1A1_L_DI_16x24VDC_ST_2 : WORD;
		R1A1_L_DI_16x24VDC_ST_3 : WORD;
		R1A1_L_DI_16x24VDC_ST_4 : WORD;
		R2A1_L_AI_4xU_I_2_wire_ST_1 : ARRAY[0..7] OF BYTE;
		R2A1_L_DI_16x24VDC_ST_1 : WORD;
		R2A1_L_DI_16x24VDC_ST_2 : WORD;
		R2A1_L_DI_16x24VDC_ST_3 : WORD;
		R2A1_L_DI_16x24VDC_ST_4 : WORD;
		R2A1_L_DI_16x24VDC_ST_5 : WORD;
		R2A1_L_DI_16x24VDC_ST_6 : WORD;
		R2A1_L_TM_Pulse_2x24V_1 : ARRAY[0..15] OF BYTE;
		R6_L_DI_16x24VDC_ST_1 : WORD;
		R6_L_DI_16x24VDC_ST_2 : WORD;
		WP002_DM260_L_Acquisition_Status_1 : ARRAY[0..2] OF BYTE;
		WP002_DM260_L_Results_Status_1 : BYTE;
		WP002_DM260_L_Soft_Event_Control_1 : BYTE;
		WP002_DM260_L_Result_Data_64_bytes_1 : ARRAY[0..71] OF BYTE;
		fx0_gpnt_L_Input_Data_Block_1_1 : ARRAY[0..11] OF BYTE;
		fx0_gpnt_L_Input_Data_Block_2_1 : ARRAY[0..11] OF BYTE;
		fx0_gpnt_L_Input_Data_Block_3_1 : ARRAY[0..11] OF BYTE;
		fx0_gpnt_L_Input_Data_Block_4_1 : ARRAY[0..11] OF BYTE;
		fx0_gpnt_L_Input_Data_Block_5_1 : WORD;
		WP004_DM260_L_Acquisition_Status_1 : ARRAY[0..2] OF BYTE;
		WP004_DM260_L_Results_Status_1 : BYTE;
		WP004_DM260_L_Soft_Event_Control_1 : BYTE;
		WP004_DM260_L_Result_Data_64_bytes_1 : ARRAY[0..71] OF BYTE;
		WP0031_DM260_L_Acquisition_Status_1 : ARRAY[0..2] OF BYTE;
		WP0031_DM260_L_Results_Status_1 : BYTE;
		WP0031_DM260_L_Soft_Event_Control_1 : BYTE;
		WP0031_DM260_L_Result_Data_64_bytes_1 : ARRAY[0..71] OF BYTE;
		WP003_DM260_L_Acquisition_Status_1 : ARRAY[0..2] OF BYTE;
		WP003_DM260_L_Results_Status_1 : BYTE;
		WP003_DM260_L_Soft_Event_Control_1 : BYTE;
		WP003_DM260_L_Result_Data_64_bytes_1 : ARRAY[0..71] OF BYTE;
		WP005_DM260_L_Acquisition_Status_1 : ARRAY[0..2] OF BYTE;
		WP005_DM260_L_Results_Status_1 : BYTE;
		WP005_DM260_L_Soft_Event_Control_1 : BYTE;
		WP005_DM260_L_Result_Data_64_bytes_1 : ARRAY[0..71] OF BYTE;
		WP006_DM260_L_Acquisition_Status_1 : ARRAY[0..2] OF BYTE;
		WP006_DM260_L_Results_Status_1 : BYTE;
		WP006_DM260_L_Soft_Event_Control_1 : BYTE;
		WP006_DM260_L_Result_Data_64_bytes_1 : ARRAY[0..71] OF BYTE;
		WP001_DM8050_L_Acquisition_Status_1 : ARRAY[0..2] OF BYTE;
		WP001_DM8050_L_Results_Status_1 : BYTE;
		WP001_DM8050_L_Soft_Event_Control_1 : BYTE;
		WP001_DM8050_L_Result_Data_64_bytes_1 : ARRAY[0..71] OF BYTE;
		WP004_DM8050_L_Acquisition_Status_1 : ARRAY[0..2] OF BYTE;
		WP004_DM8050_L_Results_Status_1 : BYTE;
		WP004_DM8050_L_Soft_Event_Control_1 : BYTE;
		WP004_DM8050_L_Result_Data_64_bytes_1 : ARRAY[0..71] OF BYTE;
		WP003_CAM_L_Acquisition_Status_1 : ARRAY[0..2] OF BYTE;
		WP003_CAM_L_Inspection_Status_1 : DWORD;
		WP003_CAM_L_Command_Control_1 : WORD;
		WP003_CAM_L_SoftEvent_Control_1 : BYTE;
		WP003_CAM_L_Results_64_bytes_1 : ARRAY[0..67] OF BYTE;
		WP004_CAM_L_Acquisition_Status_1 : ARRAY[0..2] OF BYTE;
		WP004_CAM_L_Inspection_Status_1 : DWORD;
		WP004_CAM_L_Command_Control_1 : WORD;
		WP004_CAM_L_SoftEvent_Control_1 : BYTE;
		WP004_CAM_L_Results_64_bytes_1 : ARRAY[0..67] OF BYTE;
		WP0031_DM8700_L_Acquisition_Status_1 : ARRAY[0..2] OF BYTE;
		WP0031_DM8700_L_Results_Status_1 : BYTE;
		WP0031_DM8700_L_Soft_Event_Control_1 : BYTE;
		WP0031_DM8700_L_Result_Data_64_bytes_1 : ARRAY[0..71] OF BYTE;
		WP002_DM8050_L_Acquisition_Status_1 : ARRAY[0..2] OF BYTE;
		WP002_DM8050_L_Results_Status_1 : BYTE;
		WP002_DM8050_L_Soft_Event_Control_1 : BYTE;
		WP002_DM8050_L_Result_Data_64_bytes_1 : ARRAY[0..71] OF BYTE;
		CPX_Rack_L_16DI_16DI_1 : WORD;
		CPX_Rack_L_16DI_16DI_2 : WORD;
		CPX_Rack_L_16DI_16DI_3 : WORD;
		CPX_Rack_L_16DI_16DI_4 : WORD;
		CPX_Rack_L_16DI_16DI_5 : WORD;
		WP000_DM260_L_Acquisition_Status_1 : ARRAY[0..2] OF BYTE;
		WP000_DM260_L_Results_Status_1 : BYTE;
		WP000_DM260_L_Soft_Event_Control_1 : BYTE;
		WP000_DM260_L_Result_Data_64_bytes_1 : ARRAY[0..71] OF BYTE;
		WP000_DM8050_L_Acquisition_Status_1 : ARRAY[0..2] OF BYTE;
		WP000_DM8050_L_Results_Status_1 : BYTE;
		WP000_DM8050_L_Soft_Event_Control_1 : BYTE;
		WP000_DM8050_L_Result_Data_64_bytes_1 : ARRAY[0..71] OF BYTE;
	END_STRUCT;
END_TYPE

(* ---- PlcOutputs.st ---- *)
TYPE
	PlcOutputs : STRUCT
		UR5_st4_L_8_O2T_Robot_IO : ARRAY[0..23] OF BYTE;
		UR5_st4_L_9_O2T_General_Purpose_Registers_1 : ARRAY[0..99] OF BYTE;
		UR5_st4_L_10_O2T_General_Purpose_Registers_2 : ARRAY[0..99] OF BYTE;
		WP001_DM260_L_Acquisition_Control_1 : BYTE;
		WP001_DM260_L_Results_Control_1 : BYTE;
		WP001_DM260_L_Soft_Event_Control_1 : BYTE;
		WP001_DM260_L_User_Data_64_bytes_1 : ARRAY[0..67] OF BYTE;
		R5A1_L_AQ_4xU_I_ST_1 : ARRAY[0..7] OF BYTE;
		R5A1_L_DQ_16x24VDC_0_5A_ST_1 : WORD;
		R5A1_L_DQ_16x24VDC_0_5A_ST_2 : WORD;
		R5A1_L_DQ_16x24VDC_0_5A_ST_3 : WORD;
		R5A1_L_DQ_16x24VDC_0_5A_ST_4 : WORD;
		R5A1_L_TM_Pulse_2x24V_1 : ARRAY[0..23] OF BYTE;
		R5A1_L_TM_Pulse_2x24V_2 : ARRAY[0..23] OF BYTE;
		R0_L_DQ_16x24VDC_0_5A_ST_1 : WORD;
		R0_L_DQ_16x24VDC_0_5A_ST_2 : WORD;
		R0_L_DQ_16x24VDC_0_5A_ST_3 : WORD;
		R0_L_DQ_16x24VDC_0_5A_ST_4 : WORD;
		R0_L_DQ_16x24VDC_0_5A_ST_5 : WORD;
		R1A1_L_DQ_16x24VDC_0_5A_ST_1 : WORD;
		R1A1_L_DQ_16x24VDC_0_5A_ST_2 : WORD;
		R1A1_L_DQ_16x24VDC_0_5A_ST_3 : WORD;
		R2A1_L_DQ_16x24VDC_0_5A_ST_1 : WORD;
		R2A1_L_DQ_16x24VDC_0_5A_ST_2 : WORD;
		R2A1_L_DQ_16x24VDC_0_5A_ST_3 : WORD;
		R2A1_L_TM_Pulse_2x24V_1 : ARRAY[0..23] OF BYTE;
		R6_L_DQ_16x24VDC_0_5A_ST_1 : WORD;
		R6_L_DQ_16x24VDC_0_5A_ST_2 : WORD;
		WP002_DM260_L_Acquisition_Control_1 : BYTE;
		WP002_DM260_L_Results_Control_1 : BYTE;
		WP002_DM260_L_Soft_Event_Control_1 : BYTE;
		WP002_DM260_L_User_Data_64_bytes_1 : ARRAY[0..67] OF BYTE;
		CPX_WP5_L_MPA1S_VMPA1_FB_EMS_8_8DO_1 : BYTE;
		CPX_WP5_L_MPA1S_VMPA1_FB_EMS_8_8DO_2 : BYTE;
		CPX_WP5_L_MPA1S_VMPA1_FB_EMS_8_8DO_3 : BYTE;
		CPX_TS_L_MPA2S_VMPA2_FB_EMS_4_4DO_1 : BYTE;
		CPX_TS_L_MPA2G_VMPA2_FB_EMG_4_4DO_1 : BYTE;
		CPX_TS_L_MPA1G_VMPA1_FB_EMG_8_8DO_2 : BYTE;
		CPX_TS_L_MPA1G_VMPA1_FB_EMG_8_8DO_3 : BYTE;
		CPX_TS_L_MPA1G_VMPA1_FB_EMG_8_8DO_4 : BYTE;
		CPX_TS_L_MPA1G_VMPA1_FB_EMG_8_8DO_5 : BYTE;
		CPX_TS_L_MPA1G_VMPA1_FB_EMG_8_8DO_6 : BYTE;
		CPX_WP2_L_MPA1S_VMPA1_FB_EMS_8_8DO_1 : BYTE;
		CPX_WP2_L_MPA1S_VMPA1_FB_EMS_8_8DO_2 : BYTE;
		CPX_WP2_L_MPA1S_VMPA1_FB_EMS_8_8DO_3 : BYTE;
		CPX_WP2_L_MPA1G_VMPA1_FB_EMG_8_8DO_3 : BYTE;
		fx0_gpnt_L_Output_Data_Block_1_1 : ARRAY[0..9] OF BYTE;
		fx0_gpnt_L_Output_Data_Block_2_1 : ARRAY[0..9] OF BYTE;
		fx0_gpnt_L_Output_Data_Block_3_1 : ARRAY[0..9] OF BYTE;
		fx0_gpnt_L_Output_Data_Block_4_1 : ARRAY[0..9] OF BYTE;
		fx0_gpnt_L_Output_Data_Block_5_1 : ARRAY[0..9] OF BYTE;
		WP004_DM260_L_Acquisition_Control_1 : BYTE;
		WP004_DM260_L_Results_Control_1 : BYTE;
		WP004_DM260_L_Soft_Event_Control_1 : BYTE;
		WP004_DM260_L_User_Data_64_bytes_1 : ARRAY[0..67] OF BYTE;
		WP0031_DM260_L_Acquisition_Control_1 : BYTE;
		WP0031_DM260_L_Results_Control_1 : BYTE;
		WP0031_DM260_L_Soft_Event_Control_1 : BYTE;
		WP0031_DM260_L_User_Data_64_bytes_1 : ARRAY[0..67] OF BYTE;
		WP003_DM260_L_Acquisition_Control_1 : BYTE;
		WP003_DM260_L_Results_Control_1 : BYTE;
		WP003_DM260_L_Soft_Event_Control_1 : BYTE;
		WP003_DM260_L_User_Data_64_bytes_1 : ARRAY[0..67] OF BYTE;
		WP005_DM260_L_Acquisition_Control_1 : BYTE;
		WP005_DM260_L_Results_Control_1 : BYTE;
		WP005_DM260_L_Soft_Event_Control_1 : BYTE;
		WP005_DM260_L_User_Data_64_bytes_1 : ARRAY[0..67] OF BYTE;
		WP006_DM260_L_Acquisition_Control_1 : BYTE;
		WP006_DM260_L_Results_Control_1 : BYTE;
		WP006_DM260_L_Soft_Event_Control_1 : BYTE;
		WP006_DM260_L_User_Data_64_bytes_1 : ARRAY[0..67] OF BYTE;
		WP001_DM8050_L_Acquisition_Control_1 : BYTE;
		WP001_DM8050_L_Results_Control_1 : BYTE;
		WP001_DM8050_L_Soft_Event_Control_1 : BYTE;
		WP001_DM8050_L_User_Data_64_bytes_1 : ARRAY[0..67] OF BYTE;
		WP004_DM8050_L_Acquisition_Control_1 : BYTE;
		WP004_DM8050_L_Results_Control_1 : BYTE;
		WP004_DM8050_L_Soft_Event_Control_1 : BYTE;
		WP004_DM8050_L_User_Data_64_bytes_1 : ARRAY[0..67] OF BYTE;
		WP003_CAM_L_Acquisition_Control_1 : BYTE;
		WP003_CAM_L_Inspection_Control_1 : BYTE;
		WP003_CAM_L_Command_Control_1 : WORD;
		WP003_CAM_L_SoftEvent_Control_1 : BYTE;
		WP003_CAM_L_User_Data_64_bytes_1 : ARRAY[0..63] OF BYTE;
		WP004_CAM_L_Acquisition_Control_1 : BYTE;
		WP004_CAM_L_Inspection_Control_1 : BYTE;
		WP004_CAM_L_Command_Control_1 : WORD;
		WP004_CAM_L_SoftEvent_Control_1 : BYTE;
		WP004_CAM_L_User_Data_64_bytes_1 : ARRAY[0..63] OF BYTE;
		WP0031_DM8700_L_Acquisition_Control_1 : BYTE;
		WP0031_DM8700_L_Results_Control_1 : BYTE;
		WP0031_DM8700_L_Soft_Event_Control_1 : BYTE;
		WP0031_DM8700_L_User_Data_64_bytes_1 : ARRAY[0..67] OF BYTE;
		WP002_DM8050_L_Acquisition_Control_1 : BYTE;
		WP002_DM8050_L_Results_Control_1 : BYTE;
		WP002_DM8050_L_Soft_Event_Control_1 : BYTE;
		WP002_DM8050_L_User_Data_64_bytes_1 : ARRAY[0..67] OF BYTE;
		CPX_Rack_L_MPA1S_VMPA1_FB_EMS_8_8DO_1 : BYTE;
		CPX_Rack_L_MPA1S_VMPA1_FB_EMS_8_8DO_2 : BYTE;
		CPX_Rack_L_MPA1S_VMPA1_FB_EMS_8_8DO_3 : BYTE;
		CPX_Rack_L_MPA1S_VMPA1_FB_EMS_8_8DO_4 : BYTE;
		CPX_Rack_L_MPA1S_VMPA1_FB_EMS_8_8DO_5 : BYTE;
		WP000_DM260_L_Acquisition_Control_1 : BYTE;
		WP000_DM260_L_Results_Control_1 : BYTE;
		WP000_DM260_L_Soft_Event_Control_1 : BYTE;
		WP000_DM260_L_User_Data_64_bytes_1 : ARRAY[0..67] OF BYTE;
		WP000_DM8050_L_Acquisition_Control_1 : BYTE;
		WP000_DM8050_L_Results_Control_1 : BYTE;
		WP000_DM8050_L_Soft_Event_Control_1 : BYTE;
		WP000_DM8050_L_User_Data_64_bytes_1 : ARRAY[0..67] OF BYTE;
	END_STRUCT;
END_TYPE
